# EPICS autosave request: specsEBE/ebe4_settings.req
$(P):1:CURRENT_MAX
$(P):1:CURRENT_STANDBY
$(P):1:EMISSION_IVAL
$(P):1:EMISSION_MAX
$(P):1:EMISSION_PMAX
$(P):1:EMISSION_PVAL
$(P):1:EMISSION_TIME_BASE
$(P):1:FLUX_IVAL
$(P):1:FLUX_MAX
$(P):1:FLUX_PVAL
$(P):1:FLUX_TIME_BASE
$(P):1:LABEL
$(P):2:CURRENT_MAX
$(P):2:CURRENT_STANDBY
$(P):2:EMISSION_IVAL
$(P):2:EMISSION_MAX
$(P):2:EMISSION_PMAX
$(P):2:EMISSION_PVAL
$(P):2:EMISSION_TIME_BASE
$(P):2:FLUX_IVAL
$(P):2:FLUX_MAX
$(P):2:FLUX_PVAL
$(P):2:FLUX_TIME_BASE
$(P):2:LABEL
$(P):3:CURRENT_MAX
$(P):3:CURRENT_STANDBY
$(P):3:EMISSION_IVAL
$(P):3:EMISSION_MAX
$(P):3:EMISSION_PMAX
$(P):3:EMISSION_PVAL
$(P):3:EMISSION_TIME_BASE
$(P):3:FLUX_IVAL
$(P):3:FLUX_MAX
$(P):3:FLUX_PVAL
$(P):3:FLUX_TIME_BASE
$(P):3:LABEL
$(P):4:CURRENT_MAX
$(P):4:CURRENT_STANDBY
$(P):4:EMISSION_IVAL
$(P):4:EMISSION_MAX
$(P):4:EMISSION_PMAX
$(P):4:EMISSION_PVAL
$(P):4:EMISSION_TIME_BASE
$(P):4:FLUX_IVAL
$(P):4:FLUX_MAX
$(P):4:FLUX_PVAL
$(P):4:FLUX_TIME_BASE
$(P):4:LABEL
$(P):VMAX
